{attribute 'GeneratedUsingTerminal: BK1250-0000-0019'}
{attribute addProperty BoxType "BK1250-0000-0019"}
{attribute addProperty Id "A_0006_CP9940_0001_40_Ch_InputKL_2EA97E3E0A_0007_CPx9xx_4_LEDs_ButtonsKL_1187B7210A_0008_CPx9xx_8_LEDs_ButtonsKL_E991A3640A_0009_CPx9xx_12_LEDs_ButtonsKL_063F09900A_0010_CPx9xx_16_LEDs_ButtonsKL_5AE00A1C0A_0011_CPx9xx_20_LEDs_ButtonsKL_CFA8830D0A_0012_CPx9xx_24_LEDs_ButtonsKL_DBC0B8440A_0013_CPx9xx_28_LEDs_ButtonsKL_6930B3B20A_0015_CPx9xx_3_2_LEDs_Buttons_InputsKL_4F0DAD840A_0016_CPx9xx_4_2_LEDs_Buttons_InputsKL_2227C35B0A_0129_KL_1002_2_Ch_Input_24V_3_0msKL1002_BB38DA8F0A_0130_CPx9xx_E_StopKL_E653A8C10A_0131_KL_1012_2_Ch_Input_24V_0_2msKL1012_BB38DA8F0A_0132_KL_1032_2_Ch_Input_48V_3_0msKL1032_BB38DA8F0A_0133_KL_1052_2_Ch_Input_24V_3_0msKL1052_BB38DA8F0A_0134_KL_1104_4_Ch_Input_24V_3_0msKL1104_4A257D2B0A_0135_KL_1114_4_Ch_Input_24V_0_2msKL1114_4A257D2B0A_0136_KL_1124_4_Ch_Input_5V_0_2msKL1124_4A257D2B0A_0137_KL_1154_4_Ch_Input_24V_3_0msKL1154_4A257D2B0A_0138_KL_1164_4_Ch_Input_24V_0_2msKL1164_4A257D2B0A_0139_KL_1184_4_Ch_Input_neg_24V_3_0msKL1184_4A257D2B0A_0140_KL_1194_4_Ch_Input_neg_24V_0_2msKL1194_4A257D2B0A_0141_KL_1212_2_Ch_Input_24V_with_PowerKL1212_EC84F46C0A_0142_KL_1232_2_Ch_Input_24V_edge_triggered_puls_expansionKL1232_BB38DA8F0A_0143_KL_1302_2_Ch_Input_24V_3_0ms_6mAKL1302_BB38DA8F0A_0144_KL_1304_4_Ch_Input_24V_3_0ms_6mAKL1304_4A257D2B0A_0145_KL_1312_2_Ch_Input_24V_0_2ms_6mAKL1312_BB38DA8F0A_0146_KL_1314_4_Ch_Input_24V_0_2ms_6mAKL1314_4A257D2B0A_0147_KL_1352_2_Ch_Input_24V_3_0ms_NAMURKL1352_B54AC54D0A_0148_KL_1362_2_Ch_Input_24V_for_break_in_alarmKL1362_B54AC54D0A_0149_KL_1382_2_Ch_Input_24V_thermistor_sensorsKL1382_B54AC54D0A_0150_KL_1402_2_Ch_Input_24V_3_0ms_type_3KL1402_BB38DA8F0A_0151_KL_1404_4_Ch_Input_24V_3_0ms_3mA_2_wireKL1404_4A257D2B0A_0152_KL_1408_8_Ch_Input_24V_3_0msKL1408_8EF4D3E90A_0153_KL_1412_2_Ch_Input_24V_0_2ms_type_3KL1412_BB38DA8F0A_0154_KL_1414_4_Ch_Input_24V_0_2ms_3mA_2_wireKL1414_4A257D2B0A_0155_KL_1418_8_Ch_Input_24V_0_2msKL1418_8EF4D3E90A_0156_KL_1434_4_Ch_Input_24V_0_2ms_6mA_2_wireKL1434_4A257D2B0A_0157_KL_1488_8_Ch_Input_24V_neg_3msKL1488_8EF4D3E90A_0158_KL_1498_8_Ch_Input_24V_neg_0_2msKL1498_8EF4D3E90A_0159_KL_1501_1_Ch_CounterKL1501_EE1D45060A_0161_KL_1501_1002KL_62DC61BC0A_0162_KL_1512_2_Ch_CounterKL1512_78388DBB0A_0163_KL_1702_2_Ch_Input_230V_10_0msKL1702_BB38DA8F0A_0164_KL_1704_4_Ch_Input_230V_10_0msKL1704_4A257D2B0A_0165_KL_1712_2_Ch_Input_120V_10_0msKL1712_BB38DA8F0A_0166_KL_1712_0060_2_Ch_Input_60V_10_0msKL_BB38DA8F0A_0167_KL_1722_2_Ch_Input_230V_10_0ms_no_power_contactsKL1722_BB38DA8F0A_0168_KL_1804_4_Ch_Input_24V_3_0ms_3_wireKL1804_4A257D2B0A_0169_KL_1808_8_Ch_Input_24V_3_0ms_2_wireKL1808_8EF4D3E90A_0170_KL_1809_16_Ch_Input_24V_3_0msKL1809_65B88BEE0A_0171_KL_1814_4_Ch_Input_24V_0_2ms_3_wireKL1814_4A257D2B0A_0172_KL_1819_16_Ch_Input_24V_0_2msKL1819_65B88BEE0A_0173_KL_1859_8_Ch_In_Output_24V_3_0ms_0_5AKL1859_C5B2A0620A_0174_KL_1862_16_Ch_Input_24V_3_0ms_flat_ribbonKL1862_65B88BEE0A_0175_KL_1862_0010_16_Ch_Input_24V_3_0ms_flat_ribbon_ground_switchingKL_65B88BEE0A_0176_KL_1872_16_Ch_Input_24V_0_2ms_flat_ribbonKL1872_65B88BEE0A_0177_KL_1889_16_Ch_Input_24V_ground_switching_3_0msKL1889_65B88BEE0A_0178_KL_1904_4_Ch_Safety_InputKL1904_7F0D69A90A_0179_KL_1908_8_Ch_Safety_InputKL1908_7F0D69A90A_0180_KM_1002_16_Ch_Input_24V_3_0msKL_65B88BEE0A_0181_KM_1004_32_Ch_Input_24V_3_0msKL_ABE340260A_0182_KM_1008_64_Ch_Input_24V_3_0msKL_E882B8F10A_0183_KM_1012_16_Ch_Input_24V_0_2msKL_65B88BEE0A_0184_KM_1014_32_Ch_Input_24V_0_2msKL_ABE340260A_0185_KM_1018_64_Ch_Input_24V_0_2msKL_E882B8F10A_0186_KM_1644_4_Ch_Input_manual_operationKL_527512750A_0187_KL_2012_2_Ch_Output_24V_0_5_AKL2012_DCA756120A_0188_KL_2022_2_Ch_Output_24V_2_0_AKL2022_DCA756120A_0189_KL_2032_2_Ch_Output_with_Protection_24V_0_5_AKL2032_DCA756120A_0190_KL_2114_4_Ch_Output_24V_0_5_AKL2114_E49EE1EF0A_0191_KL_2124_4_Ch_Output_5V_20_mAKL2124_E49EE1EF0A_0192_KL_2134_4_Ch_Output_with_Protection_24V_0_5_AKL2134_E49EE1EF0A_0193_KL_2184_4_Ch_Output_neg_24V_0_5_AKL2184_E49EE1EF0A_0194_KL_2212_2_Ch_Output_24V_0_5_A_with_DiagKL2212_BA18203A0A_0195_KL_1202_2_Ch_Input_24V_with_PowerKL1202_EC84F46C0A_0196_KL_2404_4_Ch_Output_with_Protection_24V_0_5_A_2_wireKL2404_E49EE1EF0A_0197_KL_2408_8_Ch_Output_24V_0_5_A_3_A_maxKL2408_CBAD53BF0A_0198_KL_2424_4_Ch_Output_with_Protection_24V_2_A_2_wireKL2424_E49EE1EF0A_0199_KL_2442_2_Ch_Output_24V_8_A_8_A_maxKL2442_DCA756120A_0200_KL_2488_8_Ch_Output_24V_neg_0_5_A_3_A_maxKL2488_CBAD53BF0A_0201_KL_2284_4_Ch_Output_24V_2_A_reverse_switchingKL2284_008A18FD0A_0202_KL_2502_2_Ch_PWM_Output_24VKL2502_78388DBB0A_0203_KL_2512_2_Ch_PWM_Output_24V_1_5A_negKL2512_78388DBB0A_0204_KL_2521_1_Ch_Pulse_Train_OutputKL2521_D5F341070A_0205_KL_2531_1_Ch_Stepper_24V_1_5_AKL2531_D5AE55040A_0206_KL_2531_1000_1_Ch_Stepper_24V_1_5_AKL_5C3353880A_0207_KL_2532_2_Ch_DC_Amplifier_24V_1_AKL2532_B04618740A_0208_KL_2535_2_Ch_PWM_Amplifier_24V_1_AKL2535_B04618740A_0210_KL_2541_1_Ch_Stepper_50V_5_AKL2541_D5AE55040A_0211_KL_2541_1000_1_Ch_Stepper_50V_5_AKL_5C3353880A_0212_KL_2542_2_Ch_DC_Amplifier_50V_3_5_AKL2542_B04618740A_0213_KL_2545_2_Ch_PWM_Amplifier_50V_3_5_AKL2545_B04618740A_0214_KL_2552_2_Ch_DC_Amplifier_50V_3_5_AKL2552_B04618740A_0215_KL_2602_2_Ch_Output_Relay_230V_AC_30V_DCKL2602_DCA756120A_0216_KL_2602_0010_2_Ch_Output_Relay_ZCD_230V_AC_30V_DCKL_DCA756120A_0217_KL_2612_2_Ch_Output_Relay_125V_AC_30V_DCKL2612_DCA756120A_0218_KL_2622_2_Ch_Output_Relay_230V_AC_30V_DCKL2622_DCA756120A_0219_KL_2622_0010_2_Ch_Output_Relay_ZCD_230V_AC_30V_DCKL_DCA756120A_0220_KL_2631_1_Ch_Power_Output_Relay_400V_AC_3AKL2631_DE78D3660A_0221_KL_2634_4_Ch_Power_Output_Relay_250_V_AC_30_V_DCKL2634_E49EE1EF0A_0222_KL_2641_1_Ch_Power_Output_Relay_230V_AC_16AKL2641_8487B2050A_0223_KL_2641_1_Ch_Power_Output_Relay_230V_AC_16AKL_AF699C3C0A_0224_KL_2652_2_Ch_Power_Output_Relay_230V_AC_1AKL2652_DCA756120A_0225_KL_2692_Cycle_Monitoring_TerminalKL_6148C9040A_0226_KL_2701_1_Ch_Solid_State_Load_Relay_230V_AC_3AKL2701_DE78D3660A_0227_KL_2702_2_Ch_Output_Solid_State_Relay_230V_AC_DC_0_3AKL2702_DCA756120A_0228_KL_2702_0002_2_Ch_Output_Solid_State_Relay_230V_AC_DC_2A_mutually_lockedKL_DCA756120A_0229_KL_2702_0020_2_Ch_Output_Solid_State_Relay_230V_AC_DC_1_5AKL_DCA756120A_0230_KL_2712_2_Ch_Triac_Output_12_230V_AC_0_5AKL2712_DCA756120A_0231_KL_2722_2_Ch_Triac_Output_12_230V_AC_0_01_1AKL2722_DCA756120A_0232_KL_2732_2_Ch_Triac_Output_12_230V_AC_0_01_1A_no_power_contactsKL2732_DCA756120A_0233_KL_2744_4_Ch_Output_Solid_State_Relay_230V_AC_DC_1_5AKL2744_E49EE1EF0A_0234_KL_2751_1_Ch_Universal_Dimmer_230V_AC_300VAKL2751_6148C9040A_0236_KL_2751_1200_1_Ch_Universal_Dimmer_120V_AC_300VAKL_6148C9040A_0238_KL_2761_1_Ch_Universal_Dimmer_230V_AC_600VAKL2761_6148C9040A_0240_KL_2784_4_Ch_Output_24V_AC_DC_2A_short_circut_proofKL2784_E49EE1EF0A_0241_KL_2791_1_Ch_Speed_Controller_230V_AC_100_VAKL2791_6148C9040A_0243_KL_2791_1200_1_Ch_Speed_Controller_120V_AC_100_VAKL_6148C9040A_0245_KL_2794_4_Ch_Output_24V_AC_DC_2A_potential_free_short_circut_proofKL2794_E49EE1EF0A_0246_KL_2798_8_Ch_Output_24V_AC_DC_2A_potential_free_short_circut_proofKL2798_CBAD53BF0A_0247_KL_2808_8_Ch_Output_with_Protection_24V_0_5_A_2_wireKL2808_CBAD53BF0A_0248_KL_2819_16_Ch_Output_24V_0_5_A_with_Diagnostic_complexKL2819_28D638410A_0250_KL_2828_8_Ch_Output_with_Protection_24V_2_0_A_2_wireKL2828_CBAD53BF0A_0251_KL_2809_16_Ch_Output_24V_0_5_AKL2809_F0D0C9F80A_0252_KL_2872_16_Ch_Output_flat_ribbon_cable_24V_0_5_AKL2872_F0D0C9F80A_0253_KL_2889_16_Ch_Output_24V_ground_switching_0_5_AKL2889_F0D0C9F80A_0254_KL_2904_4_Ch_Safety_OutputKL2904_7F0D69A90A_0255_KM_2002_16_Ch_Output_24V_0_5_AKL_F0D0C9F80A_0256_KM_2004_32_Ch_Output_24V_0_5_AKL_CF002DCA0A_0257_KM_2008_64_Ch_Output_24V_0_5_AKL_F7A5EEBF0A_0258_KM_2022_16_Ch_Output_24V_2_0_AKL_F0D0C9F80A_0259_KM_2042_16_Ch_Output_24V_0_5_AKL_F0D0C9F80A_0260_KM_2604_4_Ch_Output_Relay_230V_AC_30V_DC_16AKL_E49EE1EF0A_0261_KM_2614_4_Ch_Output_Relay_230V_AC_30V_DC_16AKL_E49EE1EF0A_0262_KM_2642_2_Ch_Power_Output_Relay_230V_AC_6AKL_F206FFFF0A_0263_KM_2652_2_Ch_Power_Output_Relay_230V_AC_6AKL_13ED1AE50A_0264_KM_2774_1001_4_Ch_Blinds_control_CM_Inputs_230V_AC_1AKL2774_6148C9040A_0265_KM_2774_4_Ch_Blinds_control_CM_Inputs_230V_AC_1AKL_6148C9040A_0266_Buerkert_valve_island_2_channelsKL_DCA756120A_0267_Buerkert_valve_island_4_channelsKL_E49EE1EF0A_0268_Buerkert_valve_island_8_channelsKL_CBAD53BF0A_0269_KL_3001_1_Ch_ana_Input_10V_0_10VKL3001_6148C9040A_0271_KL_3002_2_Ch_ana_Input_10V_0_10VKL3002_B04618740A_0273_KL_3011_1_Ch_ana_Input_0_20mAKL3011_6148C9040A_0275_KL_3012_2_Ch_ana_Input_0_20mAKL3012_B04618740A_0277_KL_3021_1_Ch_ana_Input_4_20mAKL3021_6148C9040A_0279_KL_3022_2_Ch_ana_Input_4_20mAKL3022_B04618740A_0281_KL_3041_1_Ch_ana_Input_with_Power_0_20mAKL3041_6148C9040A_0283_KL_3042_2_Ch_ana_Input_with_Power_0_20mAKL3042_B04618740A_0285_KL_3044_4_Ch_ana_Input_with_Power_0_20mAKL3044_8BE38B750A_0287_KL_3051_1_Ch_ana_Input_with_Power_4_20mAKL3051_6148C9040A_0289_KL_3052_2_Ch_ana_Input_with_Power_4_20mAKL3052_B04618740A_0291_KL_3054_4_Ch_ana_Input_with_Power_4_20mAKL3054_8BE38B750A_0293_KL_3061_1_Ch_ana_Input_0_10VKL3061_6148C9040A_0295_KL_3062_2_Ch_ana_Input_0_10VKL3062_B04618740A_0297_KL_3064_4_Ch_ana_Input_0_10VKL3064_8BE38B750A_0299_KL_3102_2_Ch_ana_Input_16_Bit_10VKL3102_B04618740A_0301_KL_3112_2_Ch_ana_Input_16_Bit_0_20mAKL3112_B04618740A_0303_KL_3122_2_Ch_ana_Input_16_Bit_4_20mAKL3122_B04618740A_0305_KL_3132_2_Ch_ana_Input_16_Bit_10VKL3132_B04618740A_0307_KL_3142_2_Ch_ana_Input_with_Power_16_Bit_0_20mAKL3142_78388DBB0A_0309_KL_3152_2_Ch_ana_Input_with_Power_16_Bit_4_20mAKL3152_78388DBB0A_0311_KL_3158_4_of_8_Ch_ana_Input_with_Power_4_20mAKL3158_8BE38B750A_0313_KL_3162_2_Ch_ana_Input_16_Bit_0_10VKL3162_78388DBB0A_0315_KL_3172_2_Ch_ana_Input_16_Bit_0_2VKL3172_78388DBB0A_0317_KL_3172_0500_2_Ch_ana_Input_16_Bit_0_0_5VKL_78388DBB0A_0319_KL_3172_1000_2_Ch_ana_Input_16_Bit_0_1VKL_78388DBB0A_0321_KL_3182_2_Ch_ana_Input_16_Bit_2VKL3182_B04618740A_0323_KL_3201_1_Ch_ana_Input_PT100_RTDKL3201_6148C9040A_0325_KL_3202_2_Ch_ana_Input_PT100_RTDKL3202_B04618740A_0327_KL_3204_4_Ch_ana_Input_PT100_RTDKL3204_8BE38B750A_0329_KL_3208_0010_4_of_8_Ch_ana_Input_PT1000_Ni1000_RTDKL_8BE38B750A_0331_KL_3214_4_Ch_ana_Input_PT100_RTD_3_wireKL3214_8BE38B750A_0333_KL_3222_2_Ch_ana_Input_PT100_RTD_high_precisionKL3222_B04618740A_0335_KL_3224KL3224_8BE38B750A_0337_KL_3228_4_of_8_Ch_ana_Input_PT1000_Ni1000_RTDKL3228_8BE38B750A_0339_KL_3302_2_Ch_ana_Input_ThermoKL3302_B04618740A_0341_KL_3311_1_Ch_ana_Input_Thermo_with_wire_break_recogKL3311_6148C9040A_0343_KL_3312_2_Ch_ana_Input_Thermo_with_wire_break_recogKL3312_B04618740A_0345_KL_3314_4_Ch_ana_Input_Thermo_with_wire_break_recogKL3314_8BE38B750A_0347_KL_3351_1_Ch_Resistor_BridgeKL3351_33637CB00A_0350_KL_3351_0001_1_Ch_Resistor_BridgeKL_C7B8B3CA0A_0353_KL_3356_1_Ch_precise_Resistor_BridgeKL3356_E004D4E20A_0356_KL_3361_1_Ch_OscilloscopeKL_EE1D45060A_0358_KL_3361_1001_1_Ch_OscilloscopeKL3361_73CB82BA0A_0359_KL_3361_1002_1_Ch_OscilloscopeKL_73CB82BA0A_0360_KL_3361_1004_1_Ch_OscilloscopeKL_73CB82BA0A_0361_KL_3361_1005_1_Ch_OscilloscopeKL_73CB82BA0A_0362_KL_3362_2_Ch_OscilloscopeKL3362_E98BF8F10"}
{attribute addProperty CRC "2813048234"}
{attribute addProperty Size "0"}
TYPE TcTerminals210_1BK1250_A7ABB5AA EXTENDS BK1250_A2FCADE7 :
STRUCT
	{attribute addProperty Name "A_0006_CP9940_0001_40_Ch_Input"}
	A_0006_CP9940_0001_40_Ch_Input : KL_2EA97E3E;
	{attribute addProperty Name "A_0007_CPx9xx_4_LEDs_Buttons"}
	A_0007_CPx9xx_4_LEDs_Buttons : KL_1187B721;
	{attribute addProperty Name "A_0008_CPx9xx_8_LEDs_Buttons"}
	A_0008_CPx9xx_8_LEDs_Buttons : KL_E991A364;
	{attribute addProperty Name "A_0009_CPx9xx_12_LEDs_Buttons"}
	A_0009_CPx9xx_12_LEDs_Buttons : KL_063F0990;
	{attribute addProperty Name "A_0010_CPx9xx_16_LEDs_Buttons"}
	A_0010_CPx9xx_16_LEDs_Buttons : KL_5AE00A1C;
	{attribute addProperty Name "A_0011_CPx9xx_20_LEDs_Buttons"}
	A_0011_CPx9xx_20_LEDs_Buttons : KL_CFA8830D;
	{attribute addProperty Name "A_0012_CPx9xx_24_LEDs_Buttons"}
	A_0012_CPx9xx_24_LEDs_Buttons : KL_DBC0B844;
	{attribute addProperty Name "A_0013_CPx9xx_28_LEDs_Buttons"}
	A_0013_CPx9xx_28_LEDs_Buttons : KL_6930B3B2;
	{attribute addProperty Name "A_0015_CPx9xx_3_2_LEDs_Buttons_Inputs"}
	A_0015_CPx9xx_3_2_LEDs_Buttons_Inputs : KL_4F0DAD84;
	{attribute addProperty Name "A_0016_CPx9xx_4_2_LEDs_Buttons_Inputs"}
	A_0016_CPx9xx_4_2_LEDs_Buttons_Inputs : KL_2227C35B;
	{attribute addProperty Name "A_0129_KL_1002_2_Ch_Input_24V_3_0ms"}
	A_0129_KL_1002_2_Ch_Input_24V_3_0ms : KL1002_BB38DA8F;
	{attribute addProperty Name "A_0130_CPx9xx_E_Stop"}
	A_0130_CPx9xx_E_Stop : KL_E653A8C1;
	{attribute addProperty Name "A_0131_KL_1012_2_Ch_Input_24V_0_2ms"}
	A_0131_KL_1012_2_Ch_Input_24V_0_2ms : KL1012_BB38DA8F;
	{attribute addProperty Name "A_0132_KL_1032_2_Ch_Input_48V_3_0ms"}
	A_0132_KL_1032_2_Ch_Input_48V_3_0ms : KL1032_BB38DA8F;
	{attribute addProperty Name "A_0133_KL_1052_2_Ch_Input_24V_3_0ms"}
	A_0133_KL_1052_2_Ch_Input_24V_3_0ms : KL1052_BB38DA8F;
	{attribute addProperty Name "A_0134_KL_1104_4_Ch_Input_24V_3_0ms"}
	A_0134_KL_1104_4_Ch_Input_24V_3_0ms : KL1104_4A257D2B;
	{attribute addProperty Name "A_0135_KL_1114_4_Ch_Input_24V_0_2ms"}
	A_0135_KL_1114_4_Ch_Input_24V_0_2ms : KL1114_4A257D2B;
	{attribute addProperty Name "A_0136_KL_1124_4_Ch_Input_5V_0_2ms"}
	A_0136_KL_1124_4_Ch_Input_5V_0_2ms : KL1124_4A257D2B;
	{attribute addProperty Name "A_0137_KL_1154_4_Ch_Input_24V_3_0ms"}
	A_0137_KL_1154_4_Ch_Input_24V_3_0ms : KL1154_4A257D2B;
	{attribute addProperty Name "A_0138_KL_1164_4_Ch_Input_24V_0_2ms"}
	A_0138_KL_1164_4_Ch_Input_24V_0_2ms : KL1164_4A257D2B;
	{attribute addProperty Name "A_0139_KL_1184_4_Ch_Input_neg_24V_3_0ms"}
	A_0139_KL_1184_4_Ch_Input_neg_24V_3_0ms : KL1184_4A257D2B;
	{attribute addProperty Name "A_0140_KL_1194_4_Ch_Input_neg_24V_0_2ms"}
	A_0140_KL_1194_4_Ch_Input_neg_24V_0_2ms : KL1194_4A257D2B;
	{attribute addProperty Name "A_0141_KL_1212_2_Ch_Input_24V_with_Power"}
	A_0141_KL_1212_2_Ch_Input_24V_with_Power : KL1212_EC84F46C;
	{attribute addProperty Name "A_0142_KL_1232_2_Ch_Input_24V_edge_triggered_puls_expansion"}
	A_0142_KL_1232_2_Ch_Input_24V_edge_triggered_puls_expansion : KL1232_BB38DA8F;
	{attribute addProperty Name "A_0143_KL_1302_2_Ch_Input_24V_3_0ms_6mA"}
	A_0143_KL_1302_2_Ch_Input_24V_3_0ms_6mA : KL1302_BB38DA8F;
	{attribute addProperty Name "A_0144_KL_1304_4_Ch_Input_24V_3_0ms_6mA"}
	A_0144_KL_1304_4_Ch_Input_24V_3_0ms_6mA : KL1304_4A257D2B;
	{attribute addProperty Name "A_0145_KL_1312_2_Ch_Input_24V_0_2ms_6mA"}
	A_0145_KL_1312_2_Ch_Input_24V_0_2ms_6mA : KL1312_BB38DA8F;
	{attribute addProperty Name "A_0146_KL_1314_4_Ch_Input_24V_0_2ms_6mA"}
	A_0146_KL_1314_4_Ch_Input_24V_0_2ms_6mA : KL1314_4A257D2B;
	{attribute addProperty Name "A_0147_KL_1352_2_Ch_Input_24V_3_0ms_NAMUR"}
	A_0147_KL_1352_2_Ch_Input_24V_3_0ms_NAMUR : KL1352_B54AC54D;
	{attribute addProperty Name "A_0148_KL_1362_2_Ch_Input_24V_for_break_in_alarm"}
	A_0148_KL_1362_2_Ch_Input_24V_for_break_in_alarm : KL1362_B54AC54D;
	{attribute addProperty Name "A_0149_KL_1382_2_Ch_Input_24V_thermistor_sensors"}
	A_0149_KL_1382_2_Ch_Input_24V_thermistor_sensors : KL1382_B54AC54D;
	{attribute addProperty Name "A_0150_KL_1402_2_Ch_Input_24V_3_0ms_type_3"}
	A_0150_KL_1402_2_Ch_Input_24V_3_0ms_type_3 : KL1402_BB38DA8F;
	{attribute addProperty Name "A_0151_KL_1404_4_Ch_Input_24V_3_0ms_3mA_2_wire"}
	A_0151_KL_1404_4_Ch_Input_24V_3_0ms_3mA_2_wire : KL1404_4A257D2B;
	{attribute addProperty Name "A_0152_KL_1408_8_Ch_Input_24V_3_0ms"}
	A_0152_KL_1408_8_Ch_Input_24V_3_0ms : KL1408_8EF4D3E9;
	{attribute addProperty Name "A_0153_KL_1412_2_Ch_Input_24V_0_2ms_type_3"}
	A_0153_KL_1412_2_Ch_Input_24V_0_2ms_type_3 : KL1412_BB38DA8F;
	{attribute addProperty Name "A_0154_KL_1414_4_Ch_Input_24V_0_2ms_3mA_2_wire"}
	A_0154_KL_1414_4_Ch_Input_24V_0_2ms_3mA_2_wire : KL1414_4A257D2B;
	{attribute addProperty Name "A_0155_KL_1418_8_Ch_Input_24V_0_2ms"}
	A_0155_KL_1418_8_Ch_Input_24V_0_2ms : KL1418_8EF4D3E9;
	{attribute addProperty Name "A_0156_KL_1434_4_Ch_Input_24V_0_2ms_6mA_2_wire"}
	A_0156_KL_1434_4_Ch_Input_24V_0_2ms_6mA_2_wire : KL1434_4A257D2B;
	{attribute addProperty Name "A_0157_KL_1488_8_Ch_Input_24V_neg_3ms"}
	A_0157_KL_1488_8_Ch_Input_24V_neg_3ms : KL1488_8EF4D3E9;
	{attribute addProperty Name "A_0158_KL_1498_8_Ch_Input_24V_neg_0_2ms"}
	A_0158_KL_1498_8_Ch_Input_24V_neg_0_2ms : KL1498_8EF4D3E9;
	{attribute addProperty Name "A_0159_KL_1501_1_Ch_Counter"}
	A_0159_KL_1501_1_Ch_Counter : KL1501_EE1D4506;
	{attribute addProperty Name "A_0161_KL_1501_1002"}
	A_0161_KL_1501_1002 : KL_62DC61BC;
	{attribute addProperty Name "A_0162_KL_1512_2_Ch_Counter"}
	A_0162_KL_1512_2_Ch_Counter : KL1512_78388DBB;
	{attribute addProperty Name "A_0163_KL_1702_2_Ch_Input_230V_10_0ms"}
	A_0163_KL_1702_2_Ch_Input_230V_10_0ms : KL1702_BB38DA8F;
	{attribute addProperty Name "A_0164_KL_1704_4_Ch_Input_230V_10_0ms"}
	A_0164_KL_1704_4_Ch_Input_230V_10_0ms : KL1704_4A257D2B;
	{attribute addProperty Name "A_0165_KL_1712_2_Ch_Input_120V_10_0ms"}
	A_0165_KL_1712_2_Ch_Input_120V_10_0ms : KL1712_BB38DA8F;
	{attribute addProperty Name "A_0166_KL_1712_0060_2_Ch_Input_60V_10_0ms"}
	A_0166_KL_1712_0060_2_Ch_Input_60V_10_0ms : KL_BB38DA8F;
	{attribute addProperty Name "A_0167_KL_1722_2_Ch_Input_230V_10_0ms_no_power_contacts"}
	A_0167_KL_1722_2_Ch_Input_230V_10_0ms_no_power_contacts : KL1722_BB38DA8F;
	{attribute addProperty Name "A_0168_KL_1804_4_Ch_Input_24V_3_0ms_3_wire"}
	A_0168_KL_1804_4_Ch_Input_24V_3_0ms_3_wire : KL1804_4A257D2B;
	{attribute addProperty Name "A_0169_KL_1808_8_Ch_Input_24V_3_0ms_2_wire"}
	A_0169_KL_1808_8_Ch_Input_24V_3_0ms_2_wire : KL1808_8EF4D3E9;
	{attribute addProperty Name "A_0170_KL_1809_16_Ch_Input_24V_3_0ms"}
	A_0170_KL_1809_16_Ch_Input_24V_3_0ms : KL1809_65B88BEE;
	{attribute addProperty Name "A_0171_KL_1814_4_Ch_Input_24V_0_2ms_3_wire"}
	A_0171_KL_1814_4_Ch_Input_24V_0_2ms_3_wire : KL1814_4A257D2B;
	{attribute addProperty Name "A_0172_KL_1819_16_Ch_Input_24V_0_2ms"}
	A_0172_KL_1819_16_Ch_Input_24V_0_2ms : KL1819_65B88BEE;
	{attribute addProperty Name "A_0173_KL_1859_8_Ch_In_Output_24V_3_0ms_0_5A"}
	A_0173_KL_1859_8_Ch_In_Output_24V_3_0ms_0_5A : KL1859_C5B2A062;
	{attribute addProperty Name "A_0174_KL_1862_16_Ch_Input_24V_3_0ms_flat_ribbon"}
	A_0174_KL_1862_16_Ch_Input_24V_3_0ms_flat_ribbon : KL1862_65B88BEE;
	{attribute addProperty Name "A_0175_KL_1862_0010_16_Ch_Input_24V_3_0ms_flat_ribbon_ground_switching"}
	A_0175_KL_1862_0010_16_Ch_Input_24V_3_0ms_flat_ribbon_ground_switching : KL_65B88BEE;
	{attribute addProperty Name "A_0176_KL_1872_16_Ch_Input_24V_0_2ms_flat_ribbon"}
	A_0176_KL_1872_16_Ch_Input_24V_0_2ms_flat_ribbon : KL1872_65B88BEE;
	{attribute addProperty Name "A_0177_KL_1889_16_Ch_Input_24V_ground_switching_3_0ms"}
	A_0177_KL_1889_16_Ch_Input_24V_ground_switching_3_0ms : KL1889_65B88BEE;
	{attribute addProperty Name "A_0178_KL_1904_4_Ch_Safety_Input"}
	A_0178_KL_1904_4_Ch_Safety_Input : KL1904_7F0D69A9;
	{attribute addProperty Name "A_0179_KL_1908_8_Ch_Safety_Input"}
	A_0179_KL_1908_8_Ch_Safety_Input : KL1908_7F0D69A9;
	{attribute addProperty Name "A_0180_KM_1002_16_Ch_Input_24V_3_0ms"}
	A_0180_KM_1002_16_Ch_Input_24V_3_0ms : KL_65B88BEE;
	{attribute addProperty Name "A_0181_KM_1004_32_Ch_Input_24V_3_0ms"}
	A_0181_KM_1004_32_Ch_Input_24V_3_0ms : KL_ABE34026;
	{attribute addProperty Name "A_0182_KM_1008_64_Ch_Input_24V_3_0ms"}
	A_0182_KM_1008_64_Ch_Input_24V_3_0ms : KL_E882B8F1;
	{attribute addProperty Name "A_0183_KM_1012_16_Ch_Input_24V_0_2ms"}
	A_0183_KM_1012_16_Ch_Input_24V_0_2ms : KL_65B88BEE;
	{attribute addProperty Name "A_0184_KM_1014_32_Ch_Input_24V_0_2ms"}
	A_0184_KM_1014_32_Ch_Input_24V_0_2ms : KL_ABE34026;
	{attribute addProperty Name "A_0185_KM_1018_64_Ch_Input_24V_0_2ms"}
	A_0185_KM_1018_64_Ch_Input_24V_0_2ms : KL_E882B8F1;
	{attribute addProperty Name "A_0186_KM_1644_4_Ch_Input_manual_operation"}
	A_0186_KM_1644_4_Ch_Input_manual_operation : KL_52751275;
	{attribute addProperty Name "A_0187_KL_2012_2_Ch_Output_24V_0_5_A"}
	A_0187_KL_2012_2_Ch_Output_24V_0_5_A : KL2012_DCA75612;
	{attribute addProperty Name "A_0188_KL_2022_2_Ch_Output_24V_2_0_A"}
	A_0188_KL_2022_2_Ch_Output_24V_2_0_A : KL2022_DCA75612;
	{attribute addProperty Name "A_0189_KL_2032_2_Ch_Output_with_Protection_24V_0_5_A"}
	A_0189_KL_2032_2_Ch_Output_with_Protection_24V_0_5_A : KL2032_DCA75612;
	{attribute addProperty Name "A_0190_KL_2114_4_Ch_Output_24V_0_5_A"}
	A_0190_KL_2114_4_Ch_Output_24V_0_5_A : KL2114_E49EE1EF;
	{attribute addProperty Name "A_0191_KL_2124_4_Ch_Output_5V_20_mA"}
	A_0191_KL_2124_4_Ch_Output_5V_20_mA : KL2124_E49EE1EF;
	{attribute addProperty Name "A_0192_KL_2134_4_Ch_Output_with_Protection_24V_0_5_A"}
	A_0192_KL_2134_4_Ch_Output_with_Protection_24V_0_5_A : KL2134_E49EE1EF;
	{attribute addProperty Name "A_0193_KL_2184_4_Ch_Output_neg_24V_0_5_A"}
	A_0193_KL_2184_4_Ch_Output_neg_24V_0_5_A : KL2184_E49EE1EF;
	{attribute addProperty Name "A_0194_KL_2212_2_Ch_Output_24V_0_5_A_with_Diag"}
	A_0194_KL_2212_2_Ch_Output_24V_0_5_A_with_Diag : KL2212_BA18203A;
	{attribute addProperty Name "A_0195_KL_1202_2_Ch_Input_24V_with_Power"}
	A_0195_KL_1202_2_Ch_Input_24V_with_Power : KL1202_EC84F46C;
	{attribute addProperty Name "A_0196_KL_2404_4_Ch_Output_with_Protection_24V_0_5_A_2_wire"}
	A_0196_KL_2404_4_Ch_Output_with_Protection_24V_0_5_A_2_wire : KL2404_E49EE1EF;
	{attribute addProperty Name "A_0197_KL_2408_8_Ch_Output_24V_0_5_A_3_A_max"}
	A_0197_KL_2408_8_Ch_Output_24V_0_5_A_3_A_max : KL2408_CBAD53BF;
	{attribute addProperty Name "A_0198_KL_2424_4_Ch_Output_with_Protection_24V_2_A_2_wire"}
	A_0198_KL_2424_4_Ch_Output_with_Protection_24V_2_A_2_wire : KL2424_E49EE1EF;
	{attribute addProperty Name "A_0199_KL_2442_2_Ch_Output_24V_8_A_8_A_max"}
	A_0199_KL_2442_2_Ch_Output_24V_8_A_8_A_max : KL2442_DCA75612;
	{attribute addProperty Name "A_0200_KL_2488_8_Ch_Output_24V_neg_0_5_A_3_A_max"}
	A_0200_KL_2488_8_Ch_Output_24V_neg_0_5_A_3_A_max : KL2488_CBAD53BF;
	{attribute addProperty Name "A_0201_KL_2284_4_Ch_Output_24V_2_A_reverse_switching"}
	A_0201_KL_2284_4_Ch_Output_24V_2_A_reverse_switching : KL2284_008A18FD;
	{attribute addProperty Name "A_0202_KL_2502_2_Ch_PWM_Output_24V"}
	A_0202_KL_2502_2_Ch_PWM_Output_24V : KL2502_78388DBB;
	{attribute addProperty Name "A_0203_KL_2512_2_Ch_PWM_Output_24V_1_5A_neg"}
	A_0203_KL_2512_2_Ch_PWM_Output_24V_1_5A_neg : KL2512_78388DBB;
	{attribute addProperty Name "A_0204_KL_2521_1_Ch_Pulse_Train_Output"}
	A_0204_KL_2521_1_Ch_Pulse_Train_Output : KL2521_D5F34107;
	{attribute addProperty Name "A_0205_KL_2531_1_Ch_Stepper_24V_1_5_A"}
	A_0205_KL_2531_1_Ch_Stepper_24V_1_5_A : KL2531_D5AE5504;
	{attribute addProperty Name "A_0206_KL_2531_1000_1_Ch_Stepper_24V_1_5_A"}
	A_0206_KL_2531_1000_1_Ch_Stepper_24V_1_5_A : KL_5C335388;
	{attribute addProperty Name "A_0207_KL_2532_2_Ch_DC_Amplifier_24V_1_A"}
	A_0207_KL_2532_2_Ch_DC_Amplifier_24V_1_A : KL2532_B0461874;
	{attribute addProperty Name "A_0208_KL_2535_2_Ch_PWM_Amplifier_24V_1_A"}
	A_0208_KL_2535_2_Ch_PWM_Amplifier_24V_1_A : KL2535_B0461874;
	{attribute addProperty Name "A_0210_KL_2541_1_Ch_Stepper_50V_5_A"}
	A_0210_KL_2541_1_Ch_Stepper_50V_5_A : KL2541_D5AE5504;
	{attribute addProperty Name "A_0211_KL_2541_1000_1_Ch_Stepper_50V_5_A"}
	A_0211_KL_2541_1000_1_Ch_Stepper_50V_5_A : KL_5C335388;
	{attribute addProperty Name "A_0212_KL_2542_2_Ch_DC_Amplifier_50V_3_5_A"}
	A_0212_KL_2542_2_Ch_DC_Amplifier_50V_3_5_A : KL2542_B0461874;
	{attribute addProperty Name "A_0213_KL_2545_2_Ch_PWM_Amplifier_50V_3_5_A"}
	A_0213_KL_2545_2_Ch_PWM_Amplifier_50V_3_5_A : KL2545_B0461874;
	{attribute addProperty Name "A_0214_KL_2552_2_Ch_DC_Amplifier_50V_3_5_A"}
	A_0214_KL_2552_2_Ch_DC_Amplifier_50V_3_5_A : KL2552_B0461874;
	{attribute addProperty Name "A_0215_KL_2602_2_Ch_Output_Relay_230V_AC_30V_DC"}
	A_0215_KL_2602_2_Ch_Output_Relay_230V_AC_30V_DC : KL2602_DCA75612;
	{attribute addProperty Name "A_0216_KL_2602_0010_2_Ch_Output_Relay_ZCD_230V_AC_30V_DC"}
	A_0216_KL_2602_0010_2_Ch_Output_Relay_ZCD_230V_AC_30V_DC : KL_DCA75612;
	{attribute addProperty Name "A_0217_KL_2612_2_Ch_Output_Relay_125V_AC_30V_DC"}
	A_0217_KL_2612_2_Ch_Output_Relay_125V_AC_30V_DC : KL2612_DCA75612;
	{attribute addProperty Name "A_0218_KL_2622_2_Ch_Output_Relay_230V_AC_30V_DC"}
	A_0218_KL_2622_2_Ch_Output_Relay_230V_AC_30V_DC : KL2622_DCA75612;
	{attribute addProperty Name "A_0219_KL_2622_0010_2_Ch_Output_Relay_ZCD_230V_AC_30V_DC"}
	A_0219_KL_2622_0010_2_Ch_Output_Relay_ZCD_230V_AC_30V_DC : KL_DCA75612;
	{attribute addProperty Name "A_0220_KL_2631_1_Ch_Power_Output_Relay_400V_AC_3A"}
	A_0220_KL_2631_1_Ch_Power_Output_Relay_400V_AC_3A : KL2631_DE78D366;
	{attribute addProperty Name "A_0221_KL_2634_4_Ch_Power_Output_Relay_250_V_AC_30_V_DC"}
	A_0221_KL_2634_4_Ch_Power_Output_Relay_250_V_AC_30_V_DC : KL2634_E49EE1EF;
	{attribute addProperty Name "A_0222_KL_2641_1_Ch_Power_Output_Relay_230V_AC_16A"}
	A_0222_KL_2641_1_Ch_Power_Output_Relay_230V_AC_16A : KL2641_8487B205;
	{attribute addProperty Name "A_0223_KL_2641_1_Ch_Power_Output_Relay_230V_AC_16A"}
	A_0223_KL_2641_1_Ch_Power_Output_Relay_230V_AC_16A : KL_AF699C3C;
	{attribute addProperty Name "A_0224_KL_2652_2_Ch_Power_Output_Relay_230V_AC_1A"}
	A_0224_KL_2652_2_Ch_Power_Output_Relay_230V_AC_1A : KL2652_DCA75612;
	{attribute addProperty Name "A_0225_KL_2692_Cycle_Monitoring_Terminal"}
	A_0225_KL_2692_Cycle_Monitoring_Terminal : KL_6148C904;
	{attribute addProperty Name "A_0226_KL_2701_1_Ch_Solid_State_Load_Relay_230V_AC_3A"}
	A_0226_KL_2701_1_Ch_Solid_State_Load_Relay_230V_AC_3A : KL2701_DE78D366;
	{attribute addProperty Name "A_0227_KL_2702_2_Ch_Output_Solid_State_Relay_230V_AC_DC_0_3A"}
	A_0227_KL_2702_2_Ch_Output_Solid_State_Relay_230V_AC_DC_0_3A : KL2702_DCA75612;
	{attribute addProperty Name "A_0228_KL_2702_0002_2_Ch_Output_Solid_State_Relay_230V_AC_DC_2A_mutually_locked"}
	A_0228_KL_2702_0002_2_Ch_Output_Solid_State_Relay_230V_AC_DC_2A_mutually_locked : KL_DCA75612;
	{attribute addProperty Name "A_0229_KL_2702_0020_2_Ch_Output_Solid_State_Relay_230V_AC_DC_1_5A"}
	A_0229_KL_2702_0020_2_Ch_Output_Solid_State_Relay_230V_AC_DC_1_5A : KL_DCA75612;
	{attribute addProperty Name "A_0230_KL_2712_2_Ch_Triac_Output_12_230V_AC_0_5A"}
	A_0230_KL_2712_2_Ch_Triac_Output_12_230V_AC_0_5A : KL2712_DCA75612;
	{attribute addProperty Name "A_0231_KL_2722_2_Ch_Triac_Output_12_230V_AC_0_01_1A"}
	A_0231_KL_2722_2_Ch_Triac_Output_12_230V_AC_0_01_1A : KL2722_DCA75612;
	{attribute addProperty Name "A_0232_KL_2732_2_Ch_Triac_Output_12_230V_AC_0_01_1A_no_power_contacts"}
	A_0232_KL_2732_2_Ch_Triac_Output_12_230V_AC_0_01_1A_no_power_contacts : KL2732_DCA75612;
	{attribute addProperty Name "A_0233_KL_2744_4_Ch_Output_Solid_State_Relay_230V_AC_DC_1_5A"}
	A_0233_KL_2744_4_Ch_Output_Solid_State_Relay_230V_AC_DC_1_5A : KL2744_E49EE1EF;
	{attribute addProperty Name "A_0234_KL_2751_1_Ch_Universal_Dimmer_230V_AC_300VA"}
	A_0234_KL_2751_1_Ch_Universal_Dimmer_230V_AC_300VA : KL2751_6148C904;
	{attribute addProperty Name "A_0236_KL_2751_1200_1_Ch_Universal_Dimmer_120V_AC_300VA"}
	A_0236_KL_2751_1200_1_Ch_Universal_Dimmer_120V_AC_300VA : KL_6148C904;
	{attribute addProperty Name "A_0238_KL_2761_1_Ch_Universal_Dimmer_230V_AC_600VA"}
	A_0238_KL_2761_1_Ch_Universal_Dimmer_230V_AC_600VA : KL2761_6148C904;
	{attribute addProperty Name "A_0240_KL_2784_4_Ch_Output_24V_AC_DC_2A_short_circut_proof"}
	A_0240_KL_2784_4_Ch_Output_24V_AC_DC_2A_short_circut_proof : KL2784_E49EE1EF;
	{attribute addProperty Name "A_0241_KL_2791_1_Ch_Speed_Controller_230V_AC_100_VA"}
	A_0241_KL_2791_1_Ch_Speed_Controller_230V_AC_100_VA : KL2791_6148C904;
	{attribute addProperty Name "A_0243_KL_2791_1200_1_Ch_Speed_Controller_120V_AC_100_VA"}
	A_0243_KL_2791_1200_1_Ch_Speed_Controller_120V_AC_100_VA : KL_6148C904;
	{attribute addProperty Name "A_0245_KL_2794_4_Ch_Output_24V_AC_DC_2A_potential_free_short_circut_proof"}
	A_0245_KL_2794_4_Ch_Output_24V_AC_DC_2A_potential_free_short_circut_proof : KL2794_E49EE1EF;
	{attribute addProperty Name "A_0246_KL_2798_8_Ch_Output_24V_AC_DC_2A_potential_free_short_circut_proof"}
	A_0246_KL_2798_8_Ch_Output_24V_AC_DC_2A_potential_free_short_circut_proof : KL2798_CBAD53BF;
	{attribute addProperty Name "A_0247_KL_2808_8_Ch_Output_with_Protection_24V_0_5_A_2_wire"}
	A_0247_KL_2808_8_Ch_Output_with_Protection_24V_0_5_A_2_wire : KL2808_CBAD53BF;
	{attribute addProperty Name "A_0248_KL_2819_16_Ch_Output_24V_0_5_A_with_Diagnostic_complex"}
	A_0248_KL_2819_16_Ch_Output_24V_0_5_A_with_Diagnostic_complex : KL2819_28D63841;
	{attribute addProperty Name "A_0250_KL_2828_8_Ch_Output_with_Protection_24V_2_0_A_2_wire"}
	A_0250_KL_2828_8_Ch_Output_with_Protection_24V_2_0_A_2_wire : KL2828_CBAD53BF;
	{attribute addProperty Name "A_0251_KL_2809_16_Ch_Output_24V_0_5_A"}
	A_0251_KL_2809_16_Ch_Output_24V_0_5_A : KL2809_F0D0C9F8;
	{attribute addProperty Name "A_0252_KL_2872_16_Ch_Output_flat_ribbon_cable_24V_0_5_A"}
	A_0252_KL_2872_16_Ch_Output_flat_ribbon_cable_24V_0_5_A : KL2872_F0D0C9F8;
	{attribute addProperty Name "A_0253_KL_2889_16_Ch_Output_24V_ground_switching_0_5_A"}
	A_0253_KL_2889_16_Ch_Output_24V_ground_switching_0_5_A : KL2889_F0D0C9F8;
	{attribute addProperty Name "A_0254_KL_2904_4_Ch_Safety_Output"}
	A_0254_KL_2904_4_Ch_Safety_Output : KL2904_7F0D69A9;
	{attribute addProperty Name "A_0255_KM_2002_16_Ch_Output_24V_0_5_A"}
	A_0255_KM_2002_16_Ch_Output_24V_0_5_A : KL_F0D0C9F8;
	{attribute addProperty Name "A_0256_KM_2004_32_Ch_Output_24V_0_5_A"}
	A_0256_KM_2004_32_Ch_Output_24V_0_5_A : KL_CF002DCA;
	{attribute addProperty Name "A_0257_KM_2008_64_Ch_Output_24V_0_5_A"}
	A_0257_KM_2008_64_Ch_Output_24V_0_5_A : KL_F7A5EEBF;
	{attribute addProperty Name "A_0258_KM_2022_16_Ch_Output_24V_2_0_A"}
	A_0258_KM_2022_16_Ch_Output_24V_2_0_A : KL_F0D0C9F8;
	{attribute addProperty Name "A_0259_KM_2042_16_Ch_Output_24V_0_5_A"}
	A_0259_KM_2042_16_Ch_Output_24V_0_5_A : KL_F0D0C9F8;
	{attribute addProperty Name "A_0260_KM_2604_4_Ch_Output_Relay_230V_AC_30V_DC_16A"}
	A_0260_KM_2604_4_Ch_Output_Relay_230V_AC_30V_DC_16A : KL_E49EE1EF;
	{attribute addProperty Name "A_0261_KM_2614_4_Ch_Output_Relay_230V_AC_30V_DC_16A"}
	A_0261_KM_2614_4_Ch_Output_Relay_230V_AC_30V_DC_16A : KL_E49EE1EF;
	{attribute addProperty Name "A_0262_KM_2642_2_Ch_Power_Output_Relay_230V_AC_6A"}
	A_0262_KM_2642_2_Ch_Power_Output_Relay_230V_AC_6A : KL_F206FFFF;
	{attribute addProperty Name "A_0263_KM_2652_2_Ch_Power_Output_Relay_230V_AC_6A"}
	A_0263_KM_2652_2_Ch_Power_Output_Relay_230V_AC_6A : KL_13ED1AE5;
	{attribute addProperty Name "A_0264_KM_2774_1001_4_Ch_Blinds_control_CM_Inputs_230V_AC_1A"}
	A_0264_KM_2774_1001_4_Ch_Blinds_control_CM_Inputs_230V_AC_1A : KL2774_6148C904;
	{attribute addProperty Name "A_0265_KM_2774_4_Ch_Blinds_control_CM_Inputs_230V_AC_1A"}
	A_0265_KM_2774_4_Ch_Blinds_control_CM_Inputs_230V_AC_1A : KL_6148C904;
	{attribute addProperty Name "A_0266_Buerkert_valve_island_2_channels"}
	A_0266_Buerkert_valve_island_2_channels : KL_DCA75612;
	{attribute addProperty Name "A_0267_Buerkert_valve_island_4_channels"}
	A_0267_Buerkert_valve_island_4_channels : KL_E49EE1EF;
	{attribute addProperty Name "A_0268_Buerkert_valve_island_8_channels"}
	A_0268_Buerkert_valve_island_8_channels : KL_CBAD53BF;
	{attribute addProperty Name "A_0269_KL_3001_1_Ch_ana_Input_10V_0_10V"}
	A_0269_KL_3001_1_Ch_ana_Input_10V_0_10V : KL3001_6148C904;
	{attribute addProperty Name "A_0271_KL_3002_2_Ch_ana_Input_10V_0_10V"}
	A_0271_KL_3002_2_Ch_ana_Input_10V_0_10V : KL3002_B0461874;
	{attribute addProperty Name "A_0273_KL_3011_1_Ch_ana_Input_0_20mA"}
	A_0273_KL_3011_1_Ch_ana_Input_0_20mA : KL3011_6148C904;
	{attribute addProperty Name "A_0275_KL_3012_2_Ch_ana_Input_0_20mA"}
	A_0275_KL_3012_2_Ch_ana_Input_0_20mA : KL3012_B0461874;
	{attribute addProperty Name "A_0277_KL_3021_1_Ch_ana_Input_4_20mA"}
	A_0277_KL_3021_1_Ch_ana_Input_4_20mA : KL3021_6148C904;
	{attribute addProperty Name "A_0279_KL_3022_2_Ch_ana_Input_4_20mA"}
	A_0279_KL_3022_2_Ch_ana_Input_4_20mA : KL3022_B0461874;
	{attribute addProperty Name "A_0281_KL_3041_1_Ch_ana_Input_with_Power_0_20mA"}
	A_0281_KL_3041_1_Ch_ana_Input_with_Power_0_20mA : KL3041_6148C904;
	{attribute addProperty Name "A_0283_KL_3042_2_Ch_ana_Input_with_Power_0_20mA"}
	A_0283_KL_3042_2_Ch_ana_Input_with_Power_0_20mA : KL3042_B0461874;
	{attribute addProperty Name "A_0285_KL_3044_4_Ch_ana_Input_with_Power_0_20mA"}
	A_0285_KL_3044_4_Ch_ana_Input_with_Power_0_20mA : KL3044_8BE38B75;
	{attribute addProperty Name "A_0287_KL_3051_1_Ch_ana_Input_with_Power_4_20mA"}
	A_0287_KL_3051_1_Ch_ana_Input_with_Power_4_20mA : KL3051_6148C904;
	{attribute addProperty Name "A_0289_KL_3052_2_Ch_ana_Input_with_Power_4_20mA"}
	A_0289_KL_3052_2_Ch_ana_Input_with_Power_4_20mA : KL3052_B0461874;
	{attribute addProperty Name "A_0291_KL_3054_4_Ch_ana_Input_with_Power_4_20mA"}
	A_0291_KL_3054_4_Ch_ana_Input_with_Power_4_20mA : KL3054_8BE38B75;
	{attribute addProperty Name "A_0293_KL_3061_1_Ch_ana_Input_0_10V"}
	A_0293_KL_3061_1_Ch_ana_Input_0_10V : KL3061_6148C904;
	{attribute addProperty Name "A_0295_KL_3062_2_Ch_ana_Input_0_10V"}
	A_0295_KL_3062_2_Ch_ana_Input_0_10V : KL3062_B0461874;
	{attribute addProperty Name "A_0297_KL_3064_4_Ch_ana_Input_0_10V"}
	A_0297_KL_3064_4_Ch_ana_Input_0_10V : KL3064_8BE38B75;
	{attribute addProperty Name "A_0299_KL_3102_2_Ch_ana_Input_16_Bit_10V"}
	A_0299_KL_3102_2_Ch_ana_Input_16_Bit_10V : KL3102_B0461874;
	{attribute addProperty Name "A_0301_KL_3112_2_Ch_ana_Input_16_Bit_0_20mA"}
	A_0301_KL_3112_2_Ch_ana_Input_16_Bit_0_20mA : KL3112_B0461874;
	{attribute addProperty Name "A_0303_KL_3122_2_Ch_ana_Input_16_Bit_4_20mA"}
	A_0303_KL_3122_2_Ch_ana_Input_16_Bit_4_20mA : KL3122_B0461874;
	{attribute addProperty Name "A_0305_KL_3132_2_Ch_ana_Input_16_Bit_10V"}
	A_0305_KL_3132_2_Ch_ana_Input_16_Bit_10V : KL3132_B0461874;
	{attribute addProperty Name "A_0307_KL_3142_2_Ch_ana_Input_with_Power_16_Bit_0_20mA"}
	A_0307_KL_3142_2_Ch_ana_Input_with_Power_16_Bit_0_20mA : KL3142_78388DBB;
	{attribute addProperty Name "A_0309_KL_3152_2_Ch_ana_Input_with_Power_16_Bit_4_20mA"}
	A_0309_KL_3152_2_Ch_ana_Input_with_Power_16_Bit_4_20mA : KL3152_78388DBB;
	{attribute addProperty Name "A_0311_KL_3158_4_of_8_Ch_ana_Input_with_Power_4_20mA"}
	A_0311_KL_3158_4_of_8_Ch_ana_Input_with_Power_4_20mA : KL3158_8BE38B75;
	{attribute addProperty Name "A_0313_KL_3162_2_Ch_ana_Input_16_Bit_0_10V"}
	A_0313_KL_3162_2_Ch_ana_Input_16_Bit_0_10V : KL3162_78388DBB;
	{attribute addProperty Name "A_0315_KL_3172_2_Ch_ana_Input_16_Bit_0_2V"}
	A_0315_KL_3172_2_Ch_ana_Input_16_Bit_0_2V : KL3172_78388DBB;
	{attribute addProperty Name "A_0317_KL_3172_0500_2_Ch_ana_Input_16_Bit_0_0_5V"}
	A_0317_KL_3172_0500_2_Ch_ana_Input_16_Bit_0_0_5V : KL_78388DBB;
	{attribute addProperty Name "A_0319_KL_3172_1000_2_Ch_ana_Input_16_Bit_0_1V"}
	A_0319_KL_3172_1000_2_Ch_ana_Input_16_Bit_0_1V : KL_78388DBB;
	{attribute addProperty Name "A_0321_KL_3182_2_Ch_ana_Input_16_Bit_2V"}
	A_0321_KL_3182_2_Ch_ana_Input_16_Bit_2V : KL3182_B0461874;
	{attribute addProperty Name "A_0323_KL_3201_1_Ch_ana_Input_PT100_RTD"}
	A_0323_KL_3201_1_Ch_ana_Input_PT100_RTD : KL3201_6148C904;
	{attribute addProperty Name "A_0325_KL_3202_2_Ch_ana_Input_PT100_RTD"}
	A_0325_KL_3202_2_Ch_ana_Input_PT100_RTD : KL3202_B0461874;
	{attribute addProperty Name "A_0327_KL_3204_4_Ch_ana_Input_PT100_RTD"}
	A_0327_KL_3204_4_Ch_ana_Input_PT100_RTD : KL3204_8BE38B75;
	{attribute addProperty Name "A_0329_KL_3208_0010_4_of_8_Ch_ana_Input_PT1000_Ni1000_RTD"}
	A_0329_KL_3208_0010_4_of_8_Ch_ana_Input_PT1000_Ni1000_RTD : KL_8BE38B75;
	{attribute addProperty Name "A_0331_KL_3214_4_Ch_ana_Input_PT100_RTD_3_wire"}
	A_0331_KL_3214_4_Ch_ana_Input_PT100_RTD_3_wire : KL3214_8BE38B75;
	{attribute addProperty Name "A_0333_KL_3222_2_Ch_ana_Input_PT100_RTD_high_precision"}
	A_0333_KL_3222_2_Ch_ana_Input_PT100_RTD_high_precision : KL3222_B0461874;
	{attribute addProperty Name "A_0335_KL_3224"}
	A_0335_KL_3224 : KL3224_8BE38B75;
	{attribute addProperty Name "A_0337_KL_3228_4_of_8_Ch_ana_Input_PT1000_Ni1000_RTD"}
	A_0337_KL_3228_4_of_8_Ch_ana_Input_PT1000_Ni1000_RTD : KL3228_8BE38B75;
	{attribute addProperty Name "A_0339_KL_3302_2_Ch_ana_Input_Thermo"}
	A_0339_KL_3302_2_Ch_ana_Input_Thermo : KL3302_B0461874;
	{attribute addProperty Name "A_0341_KL_3311_1_Ch_ana_Input_Thermo_with_wire_break_recog"}
	A_0341_KL_3311_1_Ch_ana_Input_Thermo_with_wire_break_recog : KL3311_6148C904;
	{attribute addProperty Name "A_0343_KL_3312_2_Ch_ana_Input_Thermo_with_wire_break_recog"}
	A_0343_KL_3312_2_Ch_ana_Input_Thermo_with_wire_break_recog : KL3312_B0461874;
	{attribute addProperty Name "A_0345_KL_3314_4_Ch_ana_Input_Thermo_with_wire_break_recog"}
	A_0345_KL_3314_4_Ch_ana_Input_Thermo_with_wire_break_recog : KL3314_8BE38B75;
	{attribute addProperty Name "A_0347_KL_3351_1_Ch_Resistor_Bridge"}
	A_0347_KL_3351_1_Ch_Resistor_Bridge : KL3351_33637CB0;
	{attribute addProperty Name "A_0350_KL_3351_0001_1_Ch_Resistor_Bridge"}
	A_0350_KL_3351_0001_1_Ch_Resistor_Bridge : KL_C7B8B3CA;
	{attribute addProperty Name "A_0353_KL_3356_1_Ch_precise_Resistor_Bridge"}
	A_0353_KL_3356_1_Ch_precise_Resistor_Bridge : KL3356_E004D4E2;
	{attribute addProperty Name "A_0356_KL_3361_1_Ch_Oscilloscope"}
	A_0356_KL_3361_1_Ch_Oscilloscope : KL_EE1D4506;
	{attribute addProperty Name "A_0358_KL_3361_1001_1_Ch_Oscilloscope"}
	A_0358_KL_3361_1001_1_Ch_Oscilloscope : KL3361_73CB82BA;
	{attribute addProperty Name "A_0359_KL_3361_1002_1_Ch_Oscilloscope"}
	A_0359_KL_3361_1002_1_Ch_Oscilloscope : KL_73CB82BA;
	{attribute addProperty Name "A_0360_KL_3361_1004_1_Ch_Oscilloscope"}
	A_0360_KL_3361_1004_1_Ch_Oscilloscope : KL_73CB82BA;
	{attribute addProperty Name "A_0361_KL_3361_1005_1_Ch_Oscilloscope"}
	A_0361_KL_3361_1005_1_Ch_Oscilloscope : KL_73CB82BA;
	{attribute addProperty Name "A_0362_KL_3362_2_Ch_Oscilloscope"}
	A_0362_KL_3362_2_Ch_Oscilloscope : KL3362_E98BF8F1;
END_STRUCT
END_TYPE

(* stored: Version 1.2.0.0, ProductVersion 3.1.4024.9
   DUT TcTerminals210_1BK1250_A7ABB5AA: Id {ac63a212-eab4-4718-af51-6d29fcaa2646} *)
